FUNCTION_BLOCK WORD_TO_BIT_V0
VAR_INPUT
	Word_in:WORD;
END_VAR
VAR_OUTPUT
	bit0:BIT;
	bit1:BIT;
	bit2:BIT;
	bit3:BIT;
	bit4:BIT;
	bit5:BIT;
	bit6:BIT;
	bit7:BIT;
	bit8:BIT;
	bit9:BIT;
	bit10:BIT;
	bit11:BIT;
	bit12:BIT;
	bit13:BIT;
	bit14:BIT;
	bit15:BIT;
END_VAR
VAR
END_VAR

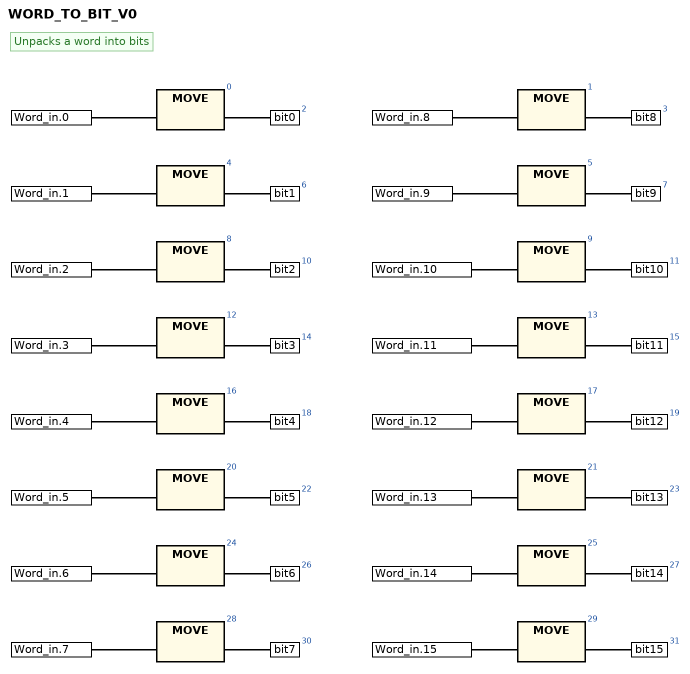
// Unpacks a word into bits
bit0 := Word_in.0;
bit8 := Word_in.8;
bit1 := Word_in.1;
bit9 := Word_in.9;
bit2 := Word_in.2;
bit10 := Word_in.10;
bit3 := Word_in.3;
bit11 := Word_in.11;
bit4 := Word_in.4;
bit12 := Word_in.12;
bit5 := Word_in.5;
bit13 := Word_in.13;
bit6 := Word_in.6;
bit14 := Word_in.14;
bit7 := Word_in.7;
bit15 := Word_in.15;

END_FUNCTION_BLOCK

(* stored: Version 1.1.0.1, ProductVersion 3.1.4024.0
   POU WORD_TO_BIT_V0: Id {e17574a5-9fe1-4a5c-824e-f1f5d9397f86}, SpecialFunc None *)
